Fanuc KAREL source: kf00078.KL

-- PROVISIONAL review KL for V940-1; original PC SHA256 a56059337c8cec41be6ce160b83dd3d83c3ca34893d6e964e767ff6e5fe3fa1a
-- Incomplete behavior may be omitted. Consult companion uncertainty JSON. Do not deploy.
PROGRAM KF00078
%NOLOCKGROUP
BEGIN
  -- V9_ZERO_TABLE_METADATA_HINT layout=0002_ascii; no indexed target words; source/name/runtime held
  -- UNRESOLVED_PC offsets 5-15; opcodes 3F,75
  -- UNRESOLVED_PC offsets 20-29; opcodes 3F,75
  -- UNRESOLVED_PC offsets 34-45; opcodes 2E,23
  -- UNRESOLVED_PC offsets 50-61; opcodes 2E,23
  -- UNRESOLVED_PC offsets 66-96; opcodes 27,22,27,2E,27,2E,22,2A,31
  -- UNRESOLVED_PC offsets 101-105; opcodes 7F
END KF00078
